(* LS Electric XG5000 project: 241002_기본회로_Yes 회로 *)
(* PLC LSPLC *)
(* module base 0 slot 0: 입력 모듈:XGI-D22A/B (DC 24V 입력, 16점 (전류소스 싱크공용/ 전류소스 입력)) *)
(* module base 0 slot 1: 출력 모듈:XGQ-RY1A (릴레이 출력, 8점 (2A용, 단독 COM.)) *)

PROGRAM NewProgram (* task: 스캔 프로그램 *)
VAR
    입력1 AT %IX0.0.0 : BOOL;
    입력10 AT %IX0.0.9 : BOOL;
    입력2 AT %IX0.0.1 : BOOL;
    입력3 AT %IX0.0.2 : BOOL;
    입력4 AT %IX0.0.3 : BOOL;
    입력5 AT %IX0.0.4 : BOOL;
    입력6 AT %IX0.0.5 : BOOL;
    입력7 AT %IX0.0.6 : BOOL;
    입력8 AT %IX0.0.7 : BOOL;
    입력9 AT %IX0.0.8 : BOOL;
    출력1 AT %QX0.1.0 : BOOL;
    출력2 AT %QX0.1.1 : BOOL;
    출력3 AT %QX0.1.2 : BOOL;
    출력4 AT %QX0.1.3 : BOOL;
    출력5 AT %QX0.1.4 : BOOL;
END_VAR

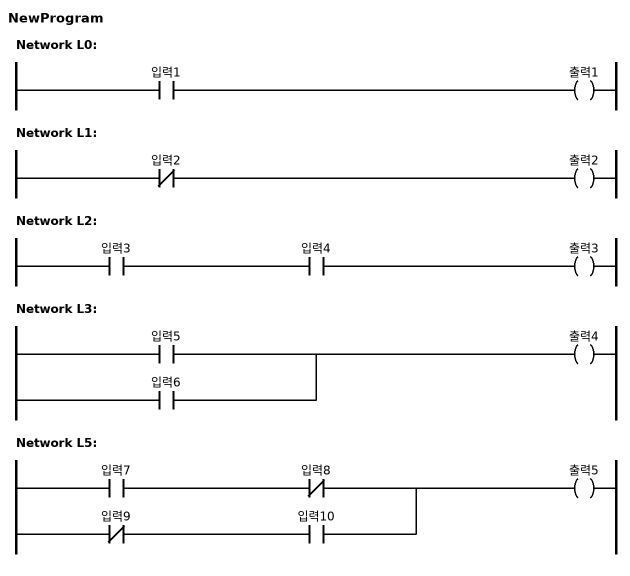
(* Rung L0 *)
출력1 := 입력1;
(* Rung L1 *)
출력2 := NOT 입력2;
(* Rung L2 *)
출력3 := 입력3 AND 입력4;
(* Rung L3 *)
출력4 := 입력5 OR 입력6;
(* Rung L5 *)
출력5 := (입력7 AND NOT 입력8) OR (NOT 입력9 AND 입력10);
END_PROGRAM